TYPE OP160_Recipe :
STRUCT
	OP160_Robo_Prog_No:INT;
END_STRUCT
END_TYPE

(* stored: Version 1.1.0.1, ProductVersion 3.1.4024.11
   DUT OP160_Recipe: Id {db564bb9-24d6-4c59-a6e4-2c874dd8c572} *)
